FUNCTION_BLOCK SLOT_PATH_SET (* Sets data for circle or line *)
  (* Standard: 61499-2 *)
  (* Version 1.0, 27-05-12, GASR, Universidade do Estado de Santa Catarina *)
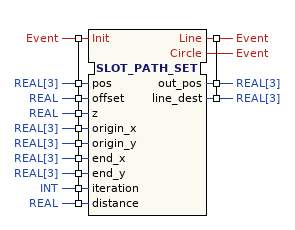
  EVENT_INPUT
    Init WITH pos, offset, z, origin_x, origin_y, end_x, end_y, iteration, distance;
  END_EVENT
  EVENT_OUTPUT
    Line WITH out_pos, line_dest;
    Circle;
  END_EVENT
  VAR_INPUT
    pos : ARRAY [0..2] OF REAL;
    offset : REAL;
    z : REAL;
    origin_x : ARRAY [0..2] OF REAL;
    origin_y : ARRAY [0..2] OF REAL;
    end_x : ARRAY [0..2] OF REAL;
    end_y : ARRAY [0..2] OF REAL;
    iteration : INT;
    distance : REAL;
  END_VAR
  VAR_OUTPUT
    out_pos : ARRAY [0..2] OF REAL;
    line_dest : ARRAY [0..2] OF REAL;
  END_VAR
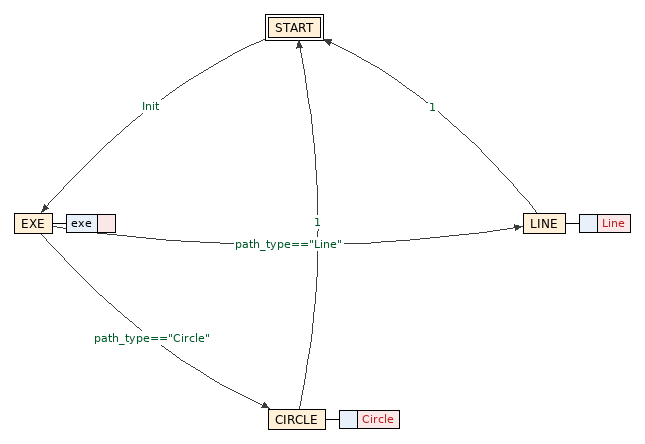
  EC_STATES
    START;
    LINE : -> Line;
    CIRCLE : -> Circle;
    EXE : exe;
  END_STATES
  EC_TRANSITIONS
    START TO EXE := Init;
    EXE TO LINE := path_type=="Line";
    EXE TO CIRCLE := path_type=="Circle";
    LINE TO START := 1;
    CIRCLE TO START := 1;
  END_TRANSITIONS
  ALGORITHM exe IN Lua:
for i = 1, 3 do
	out_pos[i] = pos[i]
	line_dest[i] = pos[i] + origin_x[i]*distance
end
  END_ALGORITHM
END_FUNCTION_BLOCK
(* other elements stored in the file *)
(* VarDeclaration Name=path_type Type=STRING *)
